// TIA Portal V16 export
// export: Created 2021-11-12T13:31:50.6360572Z, ExportSetting WithDefaults, DisplayName Totally Integrated Automation Portal, DisplayVersion V16 Update 3, DisplayName TIA Portal Version Control Interface, DisplayVersion V16 Update 2, DisplayName TIA Portal Openness, DisplayVersion V16 Update 3, DisplayName SINAMICS Startdrive Advanced, DisplayVersion V16 Update 5, DisplayName SINAMICS Startdrive G130, G150, S120, S150, SINAMICS MV, S210, DisplayVersion V16 Update 5, DisplayName SINAMICS Startdrive G110M, G120, G120C, G120D, G120P, G115D, DisplayVersion V16 Update 5, DisplayName STEP 7 Professional, DisplayVersion V16 Update 3, DisplayName STEP 7 Safety, DisplayVersion V16, DisplayName WinCC UA Professional, DisplayVersion V16 Update 3
FUNCTION_BLOCK "Cab_000+UH01"   // FB20, LAD
TITLE = FB Cabinet V1.01
{ S7_Optimized_Access := 'TRUE' }
VERSION : 0.1
// MICE Wood block
// Cabinet V1.01
// functionality regarding cabinet, like errors from main switch, circuit breakers, temperature in cabinet,……
// stored: AutoNumber false, IsIECCheckEnabled false, IsRetainMemResEnabled false, MemoryReserve 100, SetENOAutomatically false, UDAEnableTagReadback false
   VAR
      SF_FV0111_Alarm { S7_SetPoint := 'True'} : "STD_DI_Mon";
      SF_FC0114_Alarm { S7_SetPoint := 'True'} : "STD_DI_Mon";
      SF_FB0114_Alarm { S7_SetPoint := 'True'} : "STD_DI_Mon";
      "SF_I100.3_Alarm" { S7_SetPoint := 'True'} : "STD_DI_Mon";
      "SF_I100.4_Alarm" { S7_SetPoint := 'True'} : "STD_DI_Mon";
      "SF_I100.5_Alarm" { S7_SetPoint := 'True'} : "STD_DI_Mon";
      "SF_I100.6_Alarm" { S7_SetPoint := 'True'} : "STD_DI_Mon";
      "SF_I100.7_Alarm" { S7_SetPoint := 'True'} : "STD_DI_Mon";
      SF_FC2114_Alarm { S7_SetPoint := 'True'} : "STD_DI_Mon";
      SF_EC0114_Alarm { S7_SetPoint := 'True'} : "STD_DI_Mon";
      SF_FC2214_Alarm { S7_SetPoint := 'True'} : "STD_DI_Mon";
      SF_FC2314_Alarm { S7_SetPoint := 'True'} : "STD_DI_Mon";
      SF_FC2414_Alarm { S7_SetPoint := 'True'} : "STD_DI_Mon";
      SF_FC2114_Alarm_1 { S7_SetPoint := 'True'} : "STD_DI_Mon";
      SF_FC2214_Alarm_1 { S7_SetPoint := 'True'} : "STD_DI_Mon";
      "SF_I101.7_Alarm" { S7_SetPoint := 'True'} : "STD_DI_Mon";
      SF_FC3014_Alarm { S7_SetPoint := 'True'} : "STD_DI_Mon";
      SF_FC3024_Alarm { S7_SetPoint := 'True'} : "STD_DI_Mon";
      SF_RB0124_Alarm { S7_SetPoint := 'True'} : "STD_DI_Mon";
      SF_FC5014_Alarm { S7_SetPoint := 'True'} : "STD_DI_Mon";
      SF_FC5024_Alarm { S7_SetPoint := 'True'} : "STD_DI_Mon";
      "SF_I102.5_Alarm" { S7_SetPoint := 'True'} : "STD_DI_Mon";
      "SF_I102.6_Alarm" { S7_SetPoint := 'True'} : "STD_DI_Mon";
      "SF_I102.7_Alarm" { S7_SetPoint := 'True'} : "STD_DI_Mon";
   END_VAR
   VAR_TEMP
      TB1Ack : Bool;
      TB1Aux : Bool;
   END_VAR
   VAR_TEMP   // added for the SCL form of the ladder/FBD networks
      _w1 : Bool;
      _w2 : Bool;
      _w3 : Bool;
      _w4 : Bool;
      _w5 : Bool;
      _w6 : Bool;
      _w7 : Bool;
      _w8 : Bool;
      _w9 : Bool;
      _w10 : Bool;
      _w11 : Bool;
      _w12 : Bool;
   END_VAR
BEGIN

REGION Network 1: Aknowledge logic - Any zone can acknowledge alarms
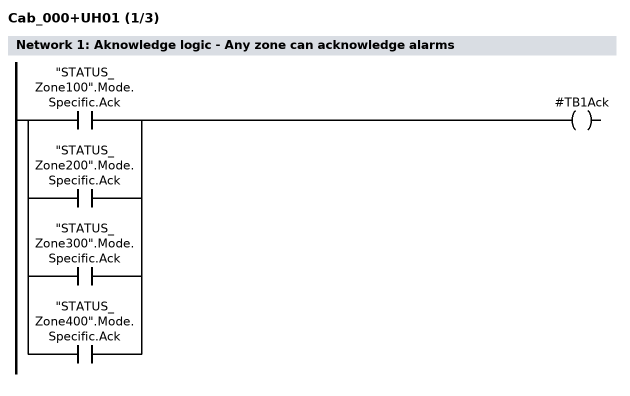
   RUNG wire#powerrail
      Contact( "STATUS_Zone100".Mode.Specific.Ack )
      wire#w1
      Coil( #TB1Ack )
   END_RUNG
   RUNG wire#powerrail
      Contact( "STATUS_Zone200".Mode.Specific.Ack )
   END_RUNG wire#w1
   RUNG wire#powerrail
      Contact( "STATUS_Zone300".Mode.Specific.Ack )
   END_RUNG wire#w1
   RUNG wire#powerrail
      Contact( "STATUS_Zone400".Mode.Specific.Ack )
   END_RUNG wire#w1
   // the same network as SCL:
   #TB1Ack := "STATUS_Zone100".Mode.Specific.Ack OR "STATUS_Zone200".Mode.Specific.Ack OR "STATUS_Zone300".Mode.Specific.Ack OR "STATUS_Zone400".Mode.Specific.Ack;
END_REGION

REGION Network 2: ************************* Alarms ******************************
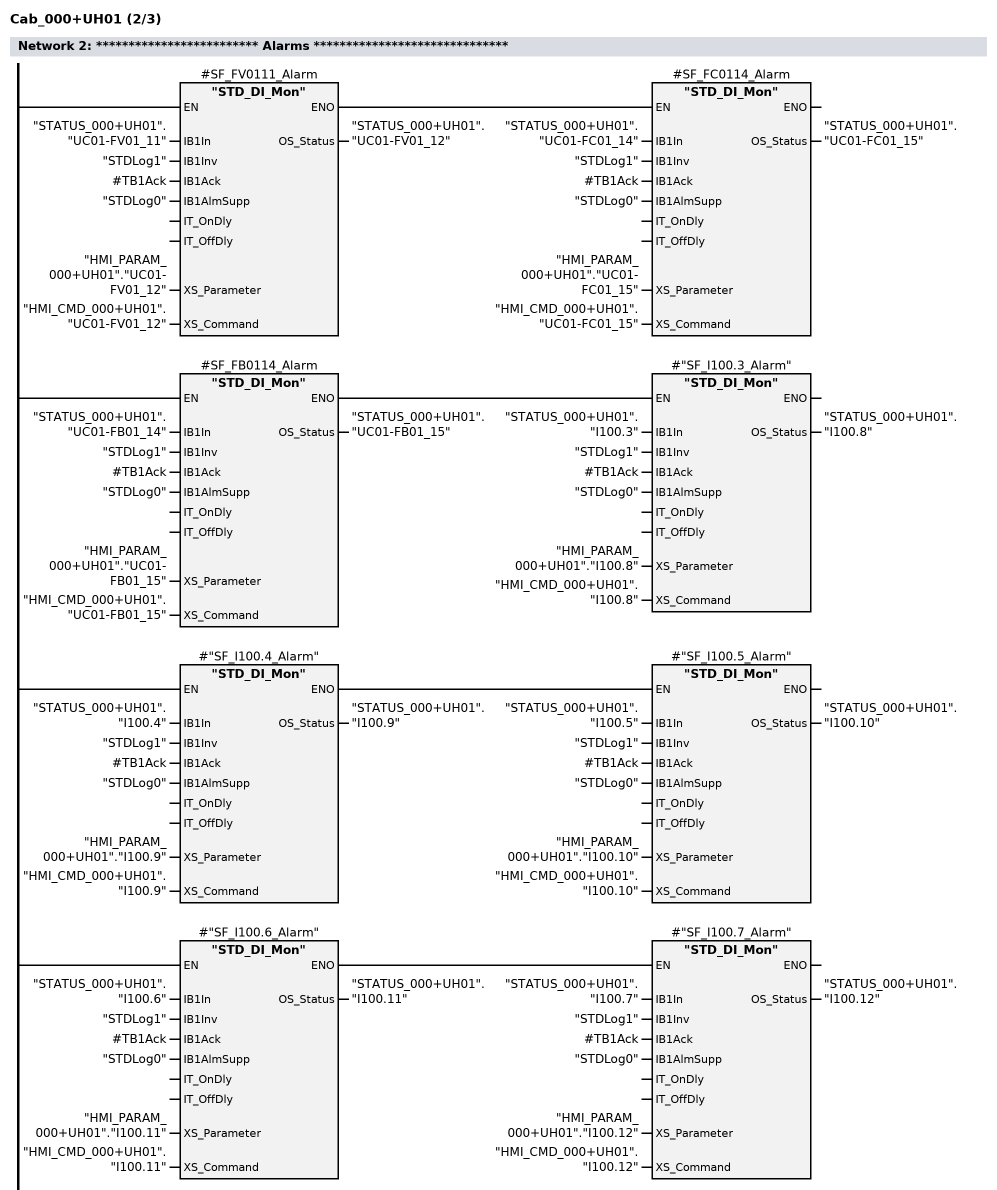
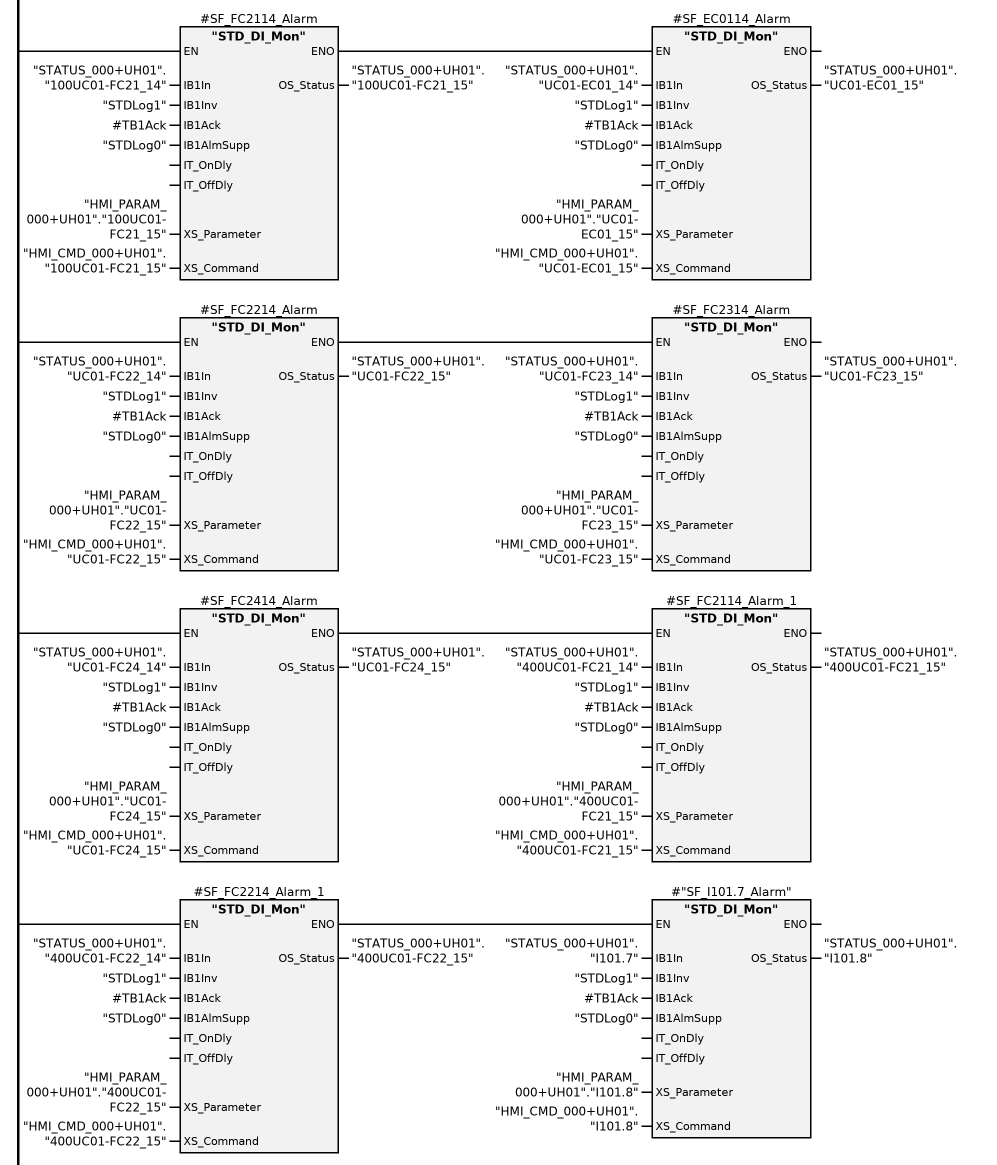
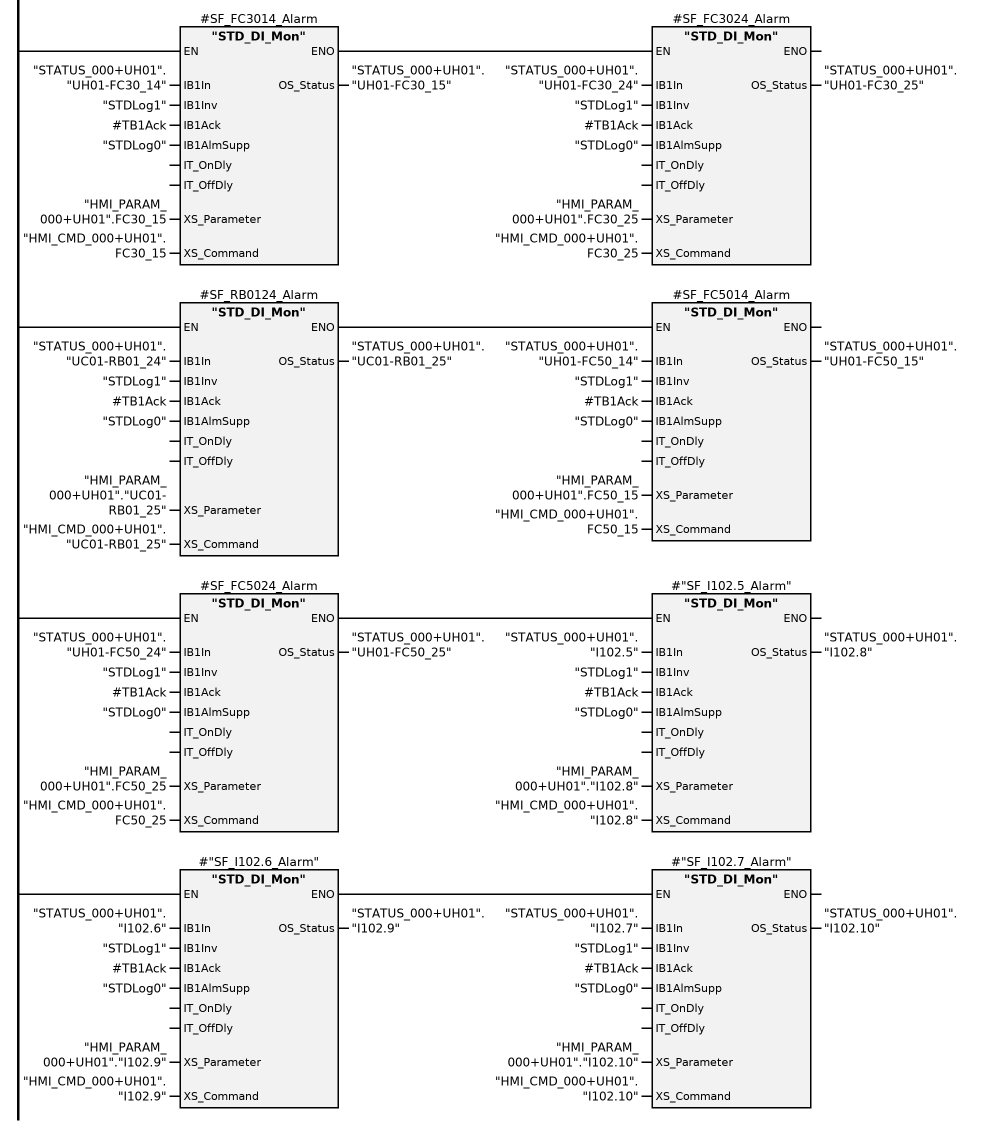
   RUNG wire#powerrail
      #SF_FV0111_Alarm(IB1In := "STATUS_000+UH01"."UC01-FV01_11", IB1Inv := "STDLog1", IB1Ack := #TB1Ack, IB1AlmSupp := "STDLog0", IT_OnDly :=, IT_OffDly :=, XS_Parameter := "HMI_PARAM_000+UH01"."UC01-FV01_12", XS_Command := "HMI_CMD_000+UH01"."UC01-FV01_12", OS_Status => "STATUS_000+UH01"."UC01-FV01_12")
      #SF_FC0114_Alarm(IB1In := "STATUS_000+UH01"."UC01-FC01_14", IB1Inv := "STDLog1", IB1Ack := #TB1Ack, IB1AlmSupp := "STDLog0", IT_OnDly :=, IT_OffDly :=, XS_Parameter := "HMI_PARAM_000+UH01"."UC01-FC01_15", XS_Command := "HMI_CMD_000+UH01"."UC01-FC01_15", OS_Status => "STATUS_000+UH01"."UC01-FC01_15")
   END_RUNG
   RUNG wire#powerrail
      #SF_FB0114_Alarm(IB1In := "STATUS_000+UH01"."UC01-FB01_14", IB1Inv := "STDLog1", IB1Ack := #TB1Ack, IB1AlmSupp := "STDLog0", IT_OnDly :=, IT_OffDly :=, XS_Parameter := "HMI_PARAM_000+UH01"."UC01-FB01_15", XS_Command := "HMI_CMD_000+UH01"."UC01-FB01_15", OS_Status => "STATUS_000+UH01"."UC01-FB01_15")
      #"SF_I100.3_Alarm"(IB1In := "STATUS_000+UH01"."I100.3", IB1Inv := "STDLog1", IB1Ack := #TB1Ack, IB1AlmSupp := "STDLog0", IT_OnDly :=, IT_OffDly :=, XS_Parameter := "HMI_PARAM_000+UH01"."I100.8", XS_Command := "HMI_CMD_000+UH01"."I100.8", OS_Status => "STATUS_000+UH01"."I100.8")
   END_RUNG
   RUNG wire#powerrail
      #"SF_I100.4_Alarm"(IB1In := "STATUS_000+UH01"."I100.4", IB1Inv := "STDLog1", IB1Ack := #TB1Ack, IB1AlmSupp := "STDLog0", IT_OnDly :=, IT_OffDly :=, XS_Parameter := "HMI_PARAM_000+UH01"."I100.9", XS_Command := "HMI_CMD_000+UH01"."I100.9", OS_Status => "STATUS_000+UH01"."I100.9")
      #"SF_I100.5_Alarm"(IB1In := "STATUS_000+UH01"."I100.5", IB1Inv := "STDLog1", IB1Ack := #TB1Ack, IB1AlmSupp := "STDLog0", IT_OnDly :=, IT_OffDly :=, XS_Parameter := "HMI_PARAM_000+UH01"."I100.10", XS_Command := "HMI_CMD_000+UH01"."I100.10", OS_Status => "STATUS_000+UH01"."I100.10")
   END_RUNG
   RUNG wire#powerrail
      #"SF_I100.6_Alarm"(IB1In := "STATUS_000+UH01"."I100.6", IB1Inv := "STDLog1", IB1Ack := #TB1Ack, IB1AlmSupp := "STDLog0", IT_OnDly :=, IT_OffDly :=, XS_Parameter := "HMI_PARAM_000+UH01"."I100.11", XS_Command := "HMI_CMD_000+UH01"."I100.11", OS_Status => "STATUS_000+UH01"."I100.11")
      #"SF_I100.7_Alarm"(IB1In := "STATUS_000+UH01"."I100.7", IB1Inv := "STDLog1", IB1Ack := #TB1Ack, IB1AlmSupp := "STDLog0", IT_OnDly :=, IT_OffDly :=, XS_Parameter := "HMI_PARAM_000+UH01"."I100.12", XS_Command := "HMI_CMD_000+UH01"."I100.12", OS_Status => "STATUS_000+UH01"."I100.12")
   END_RUNG
   RUNG wire#powerrail
      #SF_FC2114_Alarm(IB1In := "STATUS_000+UH01"."100UC01-FC21_14", IB1Inv := "STDLog1", IB1Ack := #TB1Ack, IB1AlmSupp := "STDLog0", IT_OnDly :=, IT_OffDly :=, XS_Parameter := "HMI_PARAM_000+UH01"."100UC01-FC21_15", XS_Command := "HMI_CMD_000+UH01"."100UC01-FC21_15", OS_Status => "STATUS_000+UH01"."100UC01-FC21_15")
      #SF_EC0114_Alarm(IB1In := "STATUS_000+UH01"."UC01-EC01_14", IB1Inv := "STDLog1", IB1Ack := #TB1Ack, IB1AlmSupp := "STDLog0", IT_OnDly :=, IT_OffDly :=, XS_Parameter := "HMI_PARAM_000+UH01"."UC01-EC01_15", XS_Command := "HMI_CMD_000+UH01"."UC01-EC01_15", OS_Status => "STATUS_000+UH01"."UC01-EC01_15")
   END_RUNG
   RUNG wire#powerrail
      #SF_FC2214_Alarm(IB1In := "STATUS_000+UH01"."UC01-FC22_14", IB1Inv := "STDLog1", IB1Ack := #TB1Ack, IB1AlmSupp := "STDLog0", IT_OnDly :=, IT_OffDly :=, XS_Parameter := "HMI_PARAM_000+UH01"."UC01-FC22_15", XS_Command := "HMI_CMD_000+UH01"."UC01-FC22_15", OS_Status => "STATUS_000+UH01"."UC01-FC22_15")
      #SF_FC2314_Alarm(IB1In := "STATUS_000+UH01"."UC01-FC23_14", IB1Inv := "STDLog1", IB1Ack := #TB1Ack, IB1AlmSupp := "STDLog0", IT_OnDly :=, IT_OffDly :=, XS_Parameter := "HMI_PARAM_000+UH01"."UC01-FC23_15", XS_Command := "HMI_CMD_000+UH01"."UC01-FC23_15", OS_Status => "STATUS_000+UH01"."UC01-FC23_15")
   END_RUNG
   RUNG wire#powerrail
      #SF_FC2414_Alarm(IB1In := "STATUS_000+UH01"."UC01-FC24_14", IB1Inv := "STDLog1", IB1Ack := #TB1Ack, IB1AlmSupp := "STDLog0", IT_OnDly :=, IT_OffDly :=, XS_Parameter := "HMI_PARAM_000+UH01"."UC01-FC24_15", XS_Command := "HMI_CMD_000+UH01"."UC01-FC24_15", OS_Status => "STATUS_000+UH01"."UC01-FC24_15")
      #SF_FC2114_Alarm_1(IB1In := "STATUS_000+UH01"."400UC01-FC21_14", IB1Inv := "STDLog1", IB1Ack := #TB1Ack, IB1AlmSupp := "STDLog0", IT_OnDly :=, IT_OffDly :=, XS_Parameter := "HMI_PARAM_000+UH01"."400UC01-FC21_15", XS_Command := "HMI_CMD_000+UH01"."400UC01-FC21_15", OS_Status => "STATUS_000+UH01"."400UC01-FC21_15")
   END_RUNG
   RUNG wire#powerrail
      #SF_FC2214_Alarm_1(IB1In := "STATUS_000+UH01"."400UC01-FC22_14", IB1Inv := "STDLog1", IB1Ack := #TB1Ack, IB1AlmSupp := "STDLog0", IT_OnDly :=, IT_OffDly :=, XS_Parameter := "HMI_PARAM_000+UH01"."400UC01-FC22_15", XS_Command := "HMI_CMD_000+UH01"."400UC01-FC22_15", OS_Status => "STATUS_000+UH01"."400UC01-FC22_15")
      #"SF_I101.7_Alarm"(IB1In := "STATUS_000+UH01"."I101.7", IB1Inv := "STDLog1", IB1Ack := #TB1Ack, IB1AlmSupp := "STDLog0", IT_OnDly :=, IT_OffDly :=, XS_Parameter := "HMI_PARAM_000+UH01"."I101.8", XS_Command := "HMI_CMD_000+UH01"."I101.8", OS_Status => "STATUS_000+UH01"."I101.8")
   END_RUNG
   RUNG wire#powerrail
      #SF_FC3014_Alarm(IB1In := "STATUS_000+UH01"."UH01-FC30_14", IB1Inv := "STDLog1", IB1Ack := #TB1Ack, IB1AlmSupp := "STDLog0", IT_OnDly :=, IT_OffDly :=, XS_Parameter := "HMI_PARAM_000+UH01".FC30_15, XS_Command := "HMI_CMD_000+UH01".FC30_15, OS_Status => "STATUS_000+UH01"."UH01-FC30_15")
      #SF_FC3024_Alarm(IB1In := "STATUS_000+UH01"."UH01-FC30_24", IB1Inv := "STDLog1", IB1Ack := #TB1Ack, IB1AlmSupp := "STDLog0", IT_OnDly :=, IT_OffDly :=, XS_Parameter := "HMI_PARAM_000+UH01".FC30_25, XS_Command := "HMI_CMD_000+UH01".FC30_25, OS_Status => "STATUS_000+UH01"."UH01-FC30_25")
   END_RUNG
   RUNG wire#powerrail
      #SF_RB0124_Alarm(IB1In := "STATUS_000+UH01"."UC01-RB01_24", IB1Inv := "STDLog1", IB1Ack := #TB1Ack, IB1AlmSupp := "STDLog0", IT_OnDly :=, IT_OffDly :=, XS_Parameter := "HMI_PARAM_000+UH01"."UC01-RB01_25", XS_Command := "HMI_CMD_000+UH01"."UC01-RB01_25", OS_Status => "STATUS_000+UH01"."UC01-RB01_25")
      #SF_FC5014_Alarm(IB1In := "STATUS_000+UH01"."UH01-FC50_14", IB1Inv := "STDLog1", IB1Ack := #TB1Ack, IB1AlmSupp := "STDLog0", IT_OnDly :=, IT_OffDly :=, XS_Parameter := "HMI_PARAM_000+UH01".FC50_15, XS_Command := "HMI_CMD_000+UH01".FC50_15, OS_Status => "STATUS_000+UH01"."UH01-FC50_15")
   END_RUNG
   RUNG wire#powerrail
      #SF_FC5024_Alarm(IB1In := "STATUS_000+UH01"."UH01-FC50_24", IB1Inv := "STDLog1", IB1Ack := #TB1Ack, IB1AlmSupp := "STDLog0", IT_OnDly :=, IT_OffDly :=, XS_Parameter := "HMI_PARAM_000+UH01".FC50_25, XS_Command := "HMI_CMD_000+UH01".FC50_25, OS_Status => "STATUS_000+UH01"."UH01-FC50_25")
      #"SF_I102.5_Alarm"(IB1In := "STATUS_000+UH01"."I102.5", IB1Inv := "STDLog1", IB1Ack := #TB1Ack, IB1AlmSupp := "STDLog0", IT_OnDly :=, IT_OffDly :=, XS_Parameter := "HMI_PARAM_000+UH01"."I102.8", XS_Command := "HMI_CMD_000+UH01"."I102.8", OS_Status => "STATUS_000+UH01"."I102.8")
   END_RUNG
   RUNG wire#powerrail
      #"SF_I102.6_Alarm"(IB1In := "STATUS_000+UH01"."I102.6", IB1Inv := "STDLog1", IB1Ack := #TB1Ack, IB1AlmSupp := "STDLog0", IT_OnDly :=, IT_OffDly :=, XS_Parameter := "HMI_PARAM_000+UH01"."I102.9", XS_Command := "HMI_CMD_000+UH01"."I102.9", OS_Status => "STATUS_000+UH01"."I102.9")
      #"SF_I102.7_Alarm"(IB1In := "STATUS_000+UH01"."I102.7", IB1Inv := "STDLog1", IB1Ack := #TB1Ack, IB1AlmSupp := "STDLog0", IT_OnDly :=, IT_OffDly :=, XS_Parameter := "HMI_PARAM_000+UH01"."I102.10", XS_Command := "HMI_CMD_000+UH01"."I102.10", OS_Status => "STATUS_000+UH01"."I102.10")
   END_RUNG
   // the same network as SCL:
   #SF_FV0111_Alarm(IB1In := "STATUS_000+UH01"."UC01-FV01_11",   // "STD_DI_Mon"
                    IB1Inv := "STDLog1",
                    IB1Ack := #TB1Ack,
                    IB1AlmSupp := "STDLog0",
                    XS_Parameter := "HMI_PARAM_000+UH01"."UC01-FV01_12",
                    XS_Command := "HMI_CMD_000+UH01"."UC01-FV01_12",
                    OS_Status => "STATUS_000+UH01"."UC01-FV01_12",
                    ENO => #_w1);
   IF #_w1 THEN
       #SF_FC0114_Alarm(IB1In := "STATUS_000+UH01"."UC01-FC01_14",   // "STD_DI_Mon"
                        IB1Inv := "STDLog1",
                        IB1Ack := #TB1Ack,
                        IB1AlmSupp := "STDLog0",
                        XS_Parameter := "HMI_PARAM_000+UH01"."UC01-FC01_15",
                        XS_Command := "HMI_CMD_000+UH01"."UC01-FC01_15",
                        OS_Status => "STATUS_000+UH01"."UC01-FC01_15");
   END_IF;
   #SF_FB0114_Alarm(IB1In := "STATUS_000+UH01"."UC01-FB01_14",   // "STD_DI_Mon"
                    IB1Inv := "STDLog1",
                    IB1Ack := #TB1Ack,
                    IB1AlmSupp := "STDLog0",
                    XS_Parameter := "HMI_PARAM_000+UH01"."UC01-FB01_15",
                    XS_Command := "HMI_CMD_000+UH01"."UC01-FB01_15",
                    OS_Status => "STATUS_000+UH01"."UC01-FB01_15",
                    ENO => #_w2);
   IF #_w2 THEN
       #"SF_I100.3_Alarm"(IB1In := "STATUS_000+UH01"."I100.3",   // "STD_DI_Mon"
                          IB1Inv := "STDLog1",
                          IB1Ack := #TB1Ack,
                          IB1AlmSupp := "STDLog0",
                          XS_Parameter := "HMI_PARAM_000+UH01"."I100.8",
                          XS_Command := "HMI_CMD_000+UH01"."I100.8",
                          OS_Status => "STATUS_000+UH01"."I100.8");
   END_IF;
   #"SF_I100.4_Alarm"(IB1In := "STATUS_000+UH01"."I100.4",   // "STD_DI_Mon"
                      IB1Inv := "STDLog1",
                      IB1Ack := #TB1Ack,
                      IB1AlmSupp := "STDLog0",
                      XS_Parameter := "HMI_PARAM_000+UH01"."I100.9",
                      XS_Command := "HMI_CMD_000+UH01"."I100.9",
                      OS_Status => "STATUS_000+UH01"."I100.9",
                      ENO => #_w3);
   IF #_w3 THEN
       #"SF_I100.5_Alarm"(IB1In := "STATUS_000+UH01"."I100.5",   // "STD_DI_Mon"
                          IB1Inv := "STDLog1",
                          IB1Ack := #TB1Ack,
                          IB1AlmSupp := "STDLog0",
                          XS_Parameter := "HMI_PARAM_000+UH01"."I100.10",
                          XS_Command := "HMI_CMD_000+UH01"."I100.10",
                          OS_Status => "STATUS_000+UH01"."I100.10");
   END_IF;
   #"SF_I100.6_Alarm"(IB1In := "STATUS_000+UH01"."I100.6",   // "STD_DI_Mon"
                      IB1Inv := "STDLog1",
                      IB1Ack := #TB1Ack,
                      IB1AlmSupp := "STDLog0",
                      XS_Parameter := "HMI_PARAM_000+UH01"."I100.11",
                      XS_Command := "HMI_CMD_000+UH01"."I100.11",
                      OS_Status => "STATUS_000+UH01"."I100.11",
                      ENO => #_w4);
   IF #_w4 THEN
       #"SF_I100.7_Alarm"(IB1In := "STATUS_000+UH01"."I100.7",   // "STD_DI_Mon"
                          IB1Inv := "STDLog1",
                          IB1Ack := #TB1Ack,
                          IB1AlmSupp := "STDLog0",
                          XS_Parameter := "HMI_PARAM_000+UH01"."I100.12",
                          XS_Command := "HMI_CMD_000+UH01"."I100.12",
                          OS_Status => "STATUS_000+UH01"."I100.12");
   END_IF;
   #SF_FC2114_Alarm(IB1In := "STATUS_000+UH01"."100UC01-FC21_14",   // "STD_DI_Mon"
                    IB1Inv := "STDLog1",
                    IB1Ack := #TB1Ack,
                    IB1AlmSupp := "STDLog0",
                    XS_Parameter := "HMI_PARAM_000+UH01"."100UC01-FC21_15",
                    XS_Command := "HMI_CMD_000+UH01"."100UC01-FC21_15",
                    OS_Status => "STATUS_000+UH01"."100UC01-FC21_15",
                    ENO => #_w5);
   IF #_w5 THEN
       #SF_EC0114_Alarm(IB1In := "STATUS_000+UH01"."UC01-EC01_14",   // "STD_DI_Mon"
                        IB1Inv := "STDLog1",
                        IB1Ack := #TB1Ack,
                        IB1AlmSupp := "STDLog0",
                        XS_Parameter := "HMI_PARAM_000+UH01"."UC01-EC01_15",
                        XS_Command := "HMI_CMD_000+UH01"."UC01-EC01_15",
                        OS_Status => "STATUS_000+UH01"."UC01-EC01_15");
   END_IF;
   #SF_FC2214_Alarm(IB1In := "STATUS_000+UH01"."UC01-FC22_14",   // "STD_DI_Mon"
                    IB1Inv := "STDLog1",
                    IB1Ack := #TB1Ack,
                    IB1AlmSupp := "STDLog0",
                    XS_Parameter := "HMI_PARAM_000+UH01"."UC01-FC22_15",
                    XS_Command := "HMI_CMD_000+UH01"."UC01-FC22_15",
                    OS_Status => "STATUS_000+UH01"."UC01-FC22_15",
                    ENO => #_w6);
   IF #_w6 THEN
       #SF_FC2314_Alarm(IB1In := "STATUS_000+UH01"."UC01-FC23_14",   // "STD_DI_Mon"
                        IB1Inv := "STDLog1",
                        IB1Ack := #TB1Ack,
                        IB1AlmSupp := "STDLog0",
                        XS_Parameter := "HMI_PARAM_000+UH01"."UC01-FC23_15",
                        XS_Command := "HMI_CMD_000+UH01"."UC01-FC23_15",
                        OS_Status => "STATUS_000+UH01"."UC01-FC23_15");
   END_IF;
   #SF_FC2414_Alarm(IB1In := "STATUS_000+UH01"."UC01-FC24_14",   // "STD_DI_Mon"
                    IB1Inv := "STDLog1",
                    IB1Ack := #TB1Ack,
                    IB1AlmSupp := "STDLog0",
                    XS_Parameter := "HMI_PARAM_000+UH01"."UC01-FC24_15",
                    XS_Command := "HMI_CMD_000+UH01"."UC01-FC24_15",
                    OS_Status => "STATUS_000+UH01"."UC01-FC24_15",
                    ENO => #_w7);
   IF #_w7 THEN
       #SF_FC2114_Alarm_1(IB1In := "STATUS_000+UH01"."400UC01-FC21_14",   // "STD_DI_Mon"
                          IB1Inv := "STDLog1",
                          IB1Ack := #TB1Ack,
                          IB1AlmSupp := "STDLog0",
                          XS_Parameter := "HMI_PARAM_000+UH01"."400UC01-FC21_15",
                          XS_Command := "HMI_CMD_000+UH01"."400UC01-FC21_15",
                          OS_Status => "STATUS_000+UH01"."400UC01-FC21_15");
   END_IF;
   #SF_FC2214_Alarm_1(IB1In := "STATUS_000+UH01"."400UC01-FC22_14",   // "STD_DI_Mon"
                      IB1Inv := "STDLog1",
                      IB1Ack := #TB1Ack,
                      IB1AlmSupp := "STDLog0",
                      XS_Parameter := "HMI_PARAM_000+UH01"."400UC01-FC22_15",
                      XS_Command := "HMI_CMD_000+UH01"."400UC01-FC22_15",
                      OS_Status => "STATUS_000+UH01"."400UC01-FC22_15",
                      ENO => #_w8);
   IF #_w8 THEN
       #"SF_I101.7_Alarm"(IB1In := "STATUS_000+UH01"."I101.7",   // "STD_DI_Mon"
                          IB1Inv := "STDLog1",
                          IB1Ack := #TB1Ack,
                          IB1AlmSupp := "STDLog0",
                          XS_Parameter := "HMI_PARAM_000+UH01"."I101.8",
                          XS_Command := "HMI_CMD_000+UH01"."I101.8",
                          OS_Status => "STATUS_000+UH01"."I101.8");
   END_IF;
   #SF_FC3014_Alarm(IB1In := "STATUS_000+UH01"."UH01-FC30_14",   // "STD_DI_Mon"
                    IB1Inv := "STDLog1",
                    IB1Ack := #TB1Ack,
                    IB1AlmSupp := "STDLog0",
                    XS_Parameter := "HMI_PARAM_000+UH01".FC30_15,
                    XS_Command := "HMI_CMD_000+UH01".FC30_15,
                    OS_Status => "STATUS_000+UH01"."UH01-FC30_15",
                    ENO => #_w9);
   IF #_w9 THEN
       #SF_FC3024_Alarm(IB1In := "STATUS_000+UH01"."UH01-FC30_24",   // "STD_DI_Mon"
                        IB1Inv := "STDLog1",
                        IB1Ack := #TB1Ack,
                        IB1AlmSupp := "STDLog0",
                        XS_Parameter := "HMI_PARAM_000+UH01".FC30_25,
                        XS_Command := "HMI_CMD_000+UH01".FC30_25,
                        OS_Status => "STATUS_000+UH01"."UH01-FC30_25");
   END_IF;
   #SF_RB0124_Alarm(IB1In := "STATUS_000+UH01"."UC01-RB01_24",   // "STD_DI_Mon"
                    IB1Inv := "STDLog1",
                    IB1Ack := #TB1Ack,
                    IB1AlmSupp := "STDLog0",
                    XS_Parameter := "HMI_PARAM_000+UH01"."UC01-RB01_25",
                    XS_Command := "HMI_CMD_000+UH01"."UC01-RB01_25",
                    OS_Status => "STATUS_000+UH01"."UC01-RB01_25",
                    ENO => #_w10);
   IF #_w10 THEN
       #SF_FC5014_Alarm(IB1In := "STATUS_000+UH01"."UH01-FC50_14",   // "STD_DI_Mon"
                        IB1Inv := "STDLog1",
                        IB1Ack := #TB1Ack,
                        IB1AlmSupp := "STDLog0",
                        XS_Parameter := "HMI_PARAM_000+UH01".FC50_15,
                        XS_Command := "HMI_CMD_000+UH01".FC50_15,
                        OS_Status => "STATUS_000+UH01"."UH01-FC50_15");
   END_IF;
   #SF_FC5024_Alarm(IB1In := "STATUS_000+UH01"."UH01-FC50_24",   // "STD_DI_Mon"
                    IB1Inv := "STDLog1",
                    IB1Ack := #TB1Ack,
                    IB1AlmSupp := "STDLog0",
                    XS_Parameter := "HMI_PARAM_000+UH01".FC50_25,
                    XS_Command := "HMI_CMD_000+UH01".FC50_25,
                    OS_Status => "STATUS_000+UH01"."UH01-FC50_25",
                    ENO => #_w11);
   IF #_w11 THEN
       #"SF_I102.5_Alarm"(IB1In := "STATUS_000+UH01"."I102.5",   // "STD_DI_Mon"
                          IB1Inv := "STDLog1",
                          IB1Ack := #TB1Ack,
                          IB1AlmSupp := "STDLog0",
                          XS_Parameter := "HMI_PARAM_000+UH01"."I102.8",
                          XS_Command := "HMI_CMD_000+UH01"."I102.8",
                          OS_Status => "STATUS_000+UH01"."I102.8");
   END_IF;
   #"SF_I102.6_Alarm"(IB1In := "STATUS_000+UH01"."I102.6",   // "STD_DI_Mon"
                      IB1Inv := "STDLog1",
                      IB1Ack := #TB1Ack,
                      IB1AlmSupp := "STDLog0",
                      XS_Parameter := "HMI_PARAM_000+UH01"."I102.9",
                      XS_Command := "HMI_CMD_000+UH01"."I102.9",
                      OS_Status => "STATUS_000+UH01"."I102.9",
                      ENO => #_w12);
   IF #_w12 THEN
       #"SF_I102.7_Alarm"(IB1In := "STATUS_000+UH01"."I102.7",   // "STD_DI_Mon"
                          IB1Inv := "STDLog1",
                          IB1Ack := #TB1Ack,
                          IB1AlmSupp := "STDLog0",
                          XS_Parameter := "HMI_PARAM_000+UH01"."I102.10",
                          XS_Command := "HMI_CMD_000+UH01"."I102.10",
                          OS_Status => "STATUS_000+UH01"."I102.10");
   END_IF;
END_REGION

REGION Network 3: Sum of significant alarms
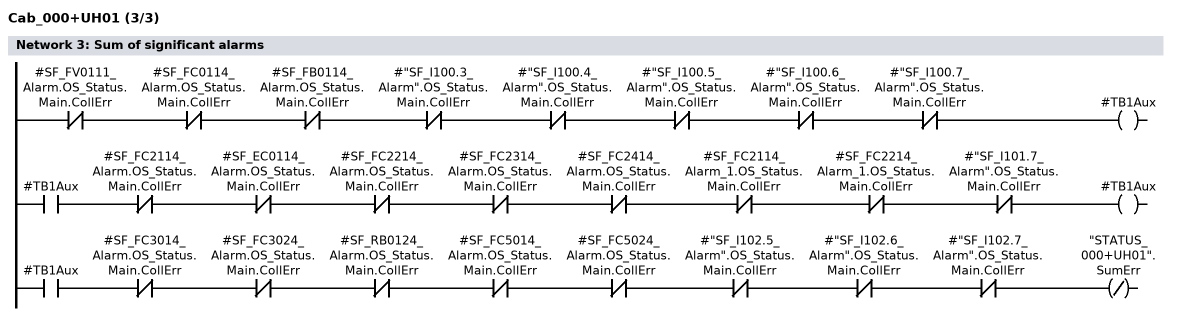
   RUNG wire#powerrail
      I_Contact( #SF_FV0111_Alarm.OS_Status.Main.CollErr )
      I_Contact( #SF_FC0114_Alarm.OS_Status.Main.CollErr )
      I_Contact( #SF_FB0114_Alarm.OS_Status.Main.CollErr )
      I_Contact( #"SF_I100.3_Alarm".OS_Status.Main.CollErr )
      I_Contact( #"SF_I100.4_Alarm".OS_Status.Main.CollErr )
      I_Contact( #"SF_I100.5_Alarm".OS_Status.Main.CollErr )
      I_Contact( #"SF_I100.6_Alarm".OS_Status.Main.CollErr )
      I_Contact( #"SF_I100.7_Alarm".OS_Status.Main.CollErr )
      Coil( #TB1Aux )
   END_RUNG
   RUNG wire#powerrail
      Contact( #TB1Aux )
      I_Contact( #SF_FC2114_Alarm.OS_Status.Main.CollErr )
      I_Contact( #SF_EC0114_Alarm.OS_Status.Main.CollErr )
      I_Contact( #SF_FC2214_Alarm.OS_Status.Main.CollErr )
      I_Contact( #SF_FC2314_Alarm.OS_Status.Main.CollErr )
      I_Contact( #SF_FC2414_Alarm.OS_Status.Main.CollErr )
      I_Contact( #SF_FC2114_Alarm_1.OS_Status.Main.CollErr )
      I_Contact( #SF_FC2214_Alarm_1.OS_Status.Main.CollErr )
      I_Contact( #"SF_I101.7_Alarm".OS_Status.Main.CollErr )
      Coil( #TB1Aux )
   END_RUNG
   RUNG wire#powerrail
      Contact( #TB1Aux )
      I_Contact( #SF_FC3014_Alarm.OS_Status.Main.CollErr )
      I_Contact( #SF_FC3024_Alarm.OS_Status.Main.CollErr )
      I_Contact( #SF_RB0124_Alarm.OS_Status.Main.CollErr )
      I_Contact( #SF_FC5014_Alarm.OS_Status.Main.CollErr )
      I_Contact( #SF_FC5024_Alarm.OS_Status.Main.CollErr )
      I_Contact( #"SF_I102.5_Alarm".OS_Status.Main.CollErr )
      I_Contact( #"SF_I102.6_Alarm".OS_Status.Main.CollErr )
      I_Contact( #"SF_I102.7_Alarm".OS_Status.Main.CollErr )
      I_Coil( "STATUS_000+UH01".SumErr )
   END_RUNG
   // the same network as SCL:
   #TB1Aux := NOT #SF_FV0111_Alarm.OS_Status.Main.CollErr AND NOT #SF_FC0114_Alarm.OS_Status.Main.CollErr AND NOT #SF_FB0114_Alarm.OS_Status.Main.CollErr AND NOT #"SF_I100.3_Alarm".OS_Status.Main.CollErr AND NOT #"SF_I100.4_Alarm".OS_Status.Main.CollErr AND NOT #"SF_I100.5_Alarm".OS_Status.Main.CollErr AND NOT #"SF_I100.6_Alarm".OS_Status.Main.CollErr AND NOT #"SF_I100.7_Alarm".OS_Status.Main.CollErr;
   #TB1Aux := #TB1Aux AND NOT #SF_FC2114_Alarm.OS_Status.Main.CollErr AND NOT #SF_EC0114_Alarm.OS_Status.Main.CollErr AND NOT #SF_FC2214_Alarm.OS_Status.Main.CollErr AND NOT #SF_FC2314_Alarm.OS_Status.Main.CollErr AND NOT #SF_FC2414_Alarm.OS_Status.Main.CollErr AND NOT #SF_FC2114_Alarm_1.OS_Status.Main.CollErr AND NOT #SF_FC2214_Alarm_1.OS_Status.Main.CollErr AND NOT #"SF_I101.7_Alarm".OS_Status.Main.CollErr;
   "STATUS_000+UH01".SumErr := NOT (#TB1Aux AND NOT #SF_FC3014_Alarm.OS_Status.Main.CollErr AND NOT #SF_FC3024_Alarm.OS_Status.Main.CollErr AND NOT #SF_RB0124_Alarm.OS_Status.Main.CollErr AND NOT #SF_FC5014_Alarm.OS_Status.Main.CollErr AND NOT #SF_FC5024_Alarm.OS_Status.Main.CollErr AND NOT #"SF_I102.5_Alarm".OS_Status.Main.CollErr AND NOT #"SF_I102.6_Alarm".OS_Status.Main.CollErr AND NOT #"SF_I102.7_Alarm".OS_Status.Main.CollErr);
END_REGION

REGION Network 4: Significant voltage OK
END_REGION
END_FUNCTION_BLOCK
